INTERFACE I_ProdManager

END_INTERFACE

(* stored: Version 1.1.0.1, ProductVersion 3.1.4024.11
   Itf I_ProdManager: Id {7fd7c27b-4c92-4e53-a24d-446ede8f376c} *)
